# EPICS autosave request: perkinElmerApp/Db/PerkinElmer_settings.req
file "ADBase_settings.req", P=$(P), R=$(R)
$(P)$(R)PECorrectionsDir
$(P)$(R)PENumOffsetFrames
$(P)$(R)PEUseOffset
$(P)$(R)PEOffsetConstant
$(P)$(R)PENumGainFrames
$(P)$(R)PEUseGain
$(P)$(R)PEGainFile
$(P)$(R)PEUsePixelCorrection
$(P)$(R)PEPixelCorrectionFile
$(P)$(R)PEGain
$(P)$(R)PESkipFrames
$(P)$(R)PENumFramesToSkip
$(P)$(R)PENumFrameBuffers
